Fanuc TP program (LS listing): MOTN023.LS

/PROG  MOTN023
/ATTR
OWNER		= MNEDITOR;
COMMENT		= "EQ EZSP2 AUF POS";
PROG_SIZE	= 753;
CREATE		= DATE 11-08-17  TIME 15:56:14;
MODIFIED	= DATE 16-05-27  TIME 06:43:26;
FILE_NAME	= ;
VERSION		= 0;
LINE_COUNT	= 13;
MEMORY_SIZE	= 1121;
PROTECT		= READ_WRITE;
TCD:  STACK_SIZE	= 0,
      TASK_PRIORITY	= 50,
      TIME_SLICE	= 0,
      BUSY_LAMP_OFF	= 0,
      ABORT_REQUEST	= 0,
      PAUSE_REQUEST	= 0;
DEFAULT_GROUP	= *,*,1,*,*;
CONTROL_CODE	= 00000000 00000000;
/MN
   1:  !EQ EZSP2 AUF POS ;
   2:  !letzte  Aenderung  31.08.2011 ;
   3:  !Ausschalten Ausgleich ;
   4:  R[820]=($MCR.$GENOVERRIDE) ;
   5:  OVERRIDE=100% ;
   6:  $SSR.$SINGLESTEP=0 ;
   7:  CALL EQGUNOPN    ;
   8:  CALL EQEND    ;
   9:  ! Open movable electrode ;
  10:  //J P[1] 100% CNT10 ACC200    ;
  11:  OVERRIDE=R[820] ;
  12:  R[819]=DO[22902]    ;
  13:  $SSR.$SINGLESTEP=R[819] ;
/POS
P[1]{
   GP3:
	UF : 1, UT : 2,
	J1=    50.000  mm
};
/END
